// TIA Portal V17 export
// export: Created 2024-09-04T07:03:07.1988734Z, ExportSetting None, DisplayName Totally Integrated Automation Portal, DisplayVersion V17 Update 7, DisplayName TIA Portal Openness, DisplayVersion V17 Update 7, DisplayName TIA Portal Version Control Interface, DisplayVersion V17, DisplayName SINAMICS Startdrive Advanced, DisplayVersion V17 SP2, DisplayName SINAMICS Startdrive G110M, G120, G120C, G120D, G120P, G115D, DisplayVersion V17 SP2, DisplayName SINAMICS Startdrive G130, G150, S120, S150, SINAMICS MV, S210, DisplayVersion V17 SP2, DisplayName STEP 7 Professional, DisplayVersion V17 Update 7, DisplayName STEP 7 Safety, DisplayVersion V17 Update 6, DisplayName WinCC Professional, DisplayVersion V17 Update 7
FUNCTION_BLOCK "fbMain"   // FB5, LAD
{ S7_Optimized_Access := 'TRUE' }
// IO processing block reads in the thermocouple and pressure transmitter readings into the program and outputs the valve control values. 
// 
// Recipe assignment waits for input from the HMI to assign recipes to each press. 
// 
// Press control FBs manage the sequencer and valve position control.
// stored: MemoryReserve 100, SetENOAutomatically false
   VAR
      iRecipeToLoad { S7_SetPoint := 'True'} : Int;
   END_VAR
   VAR CONSTANT
      iMode_ForceOpen : Int := 2;
   END_VAR
BEGIN

REGION Network 1: FB: Input/Output Processing
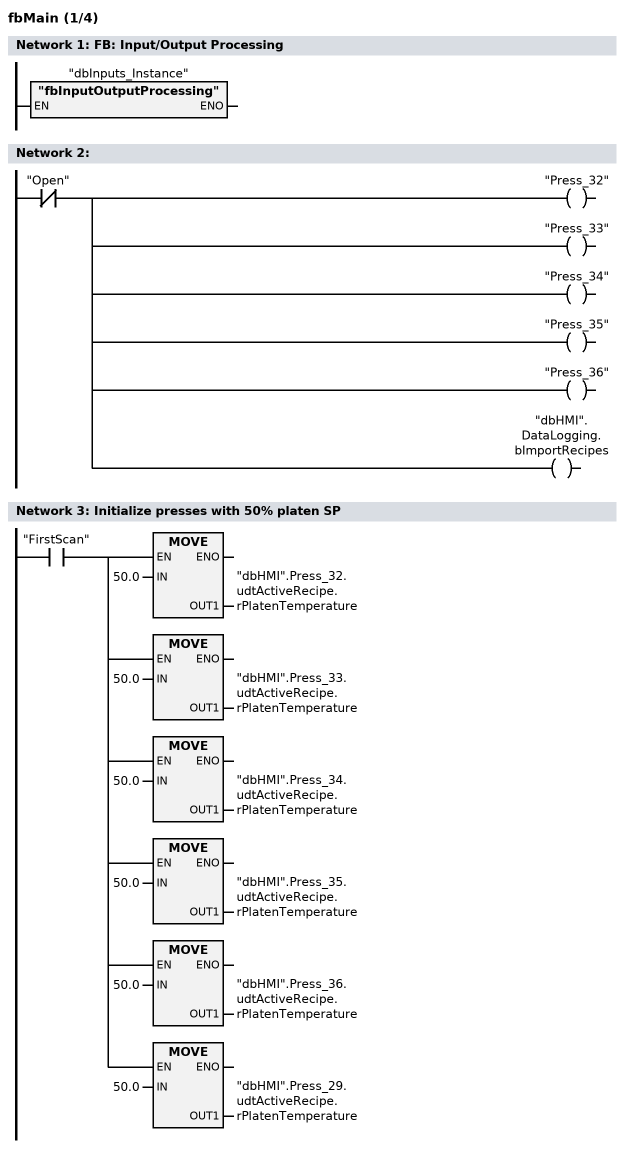
   RUNG wire#powerrail
      "dbInputs_Instance"()
   END_RUNG
   // the same network as SCL:
   "dbInputs_Instance"();   // "fbInputOutputProcessing"
END_REGION

REGION Network 2
   RUNG wire#powerrail
      I_Contact( "Open" )
      wire#w1
      Coil( "Press_32" )
   END_RUNG
   RUNG wire#w1
      Coil( "Press_33" )
   END_RUNG
   RUNG wire#w1
      Coil( "Press_34" )
   END_RUNG
   RUNG wire#w1
      Coil( "Press_35" )
   END_RUNG
   RUNG wire#w1
      Coil( "Press_36" )
   END_RUNG
   RUNG wire#w1
      Coil( "dbHMI".DataLogging.bImportRecipes )
   END_RUNG
   // the same network as SCL:
   "Press_32" := NOT "Open";
   "Press_33" := NOT "Open";
   "Press_34" := NOT "Open";
   "Press_35" := NOT "Open";
   "Press_36" := NOT "Open";
   "dbHMI".DataLogging.bImportRecipes := NOT "Open";
END_REGION

REGION Network 3: Initialize presses with 50% platen SP
   RUNG wire#powerrail
      Contact( "FirstScan" )
      wire#w1
      Move(in := 50.0, out1 => "dbHMI".Press_32.udtActiveRecipe.rPlatenTemperature)
   END_RUNG
   RUNG wire#w1
      { S7_GenerateENO := "TRUE" } Move(in := 50.0, out1 => "dbHMI".Press_33.udtActiveRecipe.rPlatenTemperature)
   END_RUNG
   RUNG wire#w1
      { S7_GenerateENO := "TRUE" } Move(in := 50.0, out1 => "dbHMI".Press_34.udtActiveRecipe.rPlatenTemperature)
   END_RUNG
   RUNG wire#w1
      { S7_GenerateENO := "TRUE" } Move(in := 50.0, out1 => "dbHMI".Press_35.udtActiveRecipe.rPlatenTemperature)
   END_RUNG
   RUNG wire#w1
      { S7_GenerateENO := "TRUE" } Move(in := 50.0, out1 => "dbHMI".Press_36.udtActiveRecipe.rPlatenTemperature)
   END_RUNG
   RUNG wire#w1
      { S7_GenerateENO := "TRUE" } Move(in := 50.0, out1 => "dbHMI".Press_29.udtActiveRecipe.rPlatenTemperature)
   END_RUNG
   // the same network as SCL:
   IF "FirstScan" THEN
       "dbHMI".Press_32.udtActiveRecipe.rPlatenTemperature := 50.0;
       "dbHMI".Press_33.udtActiveRecipe.rPlatenTemperature := 50.0;
       "dbHMI".Press_34.udtActiveRecipe.rPlatenTemperature := 50.0;
       "dbHMI".Press_35.udtActiveRecipe.rPlatenTemperature := 50.0;
       "dbHMI".Press_36.udtActiveRecipe.rPlatenTemperature := 50.0;
       "dbHMI".Press_29.udtActiveRecipe.rPlatenTemperature := 50.0;
   END_IF;
END_REGION

REGION Network 4: Initialize all presses to force open mode
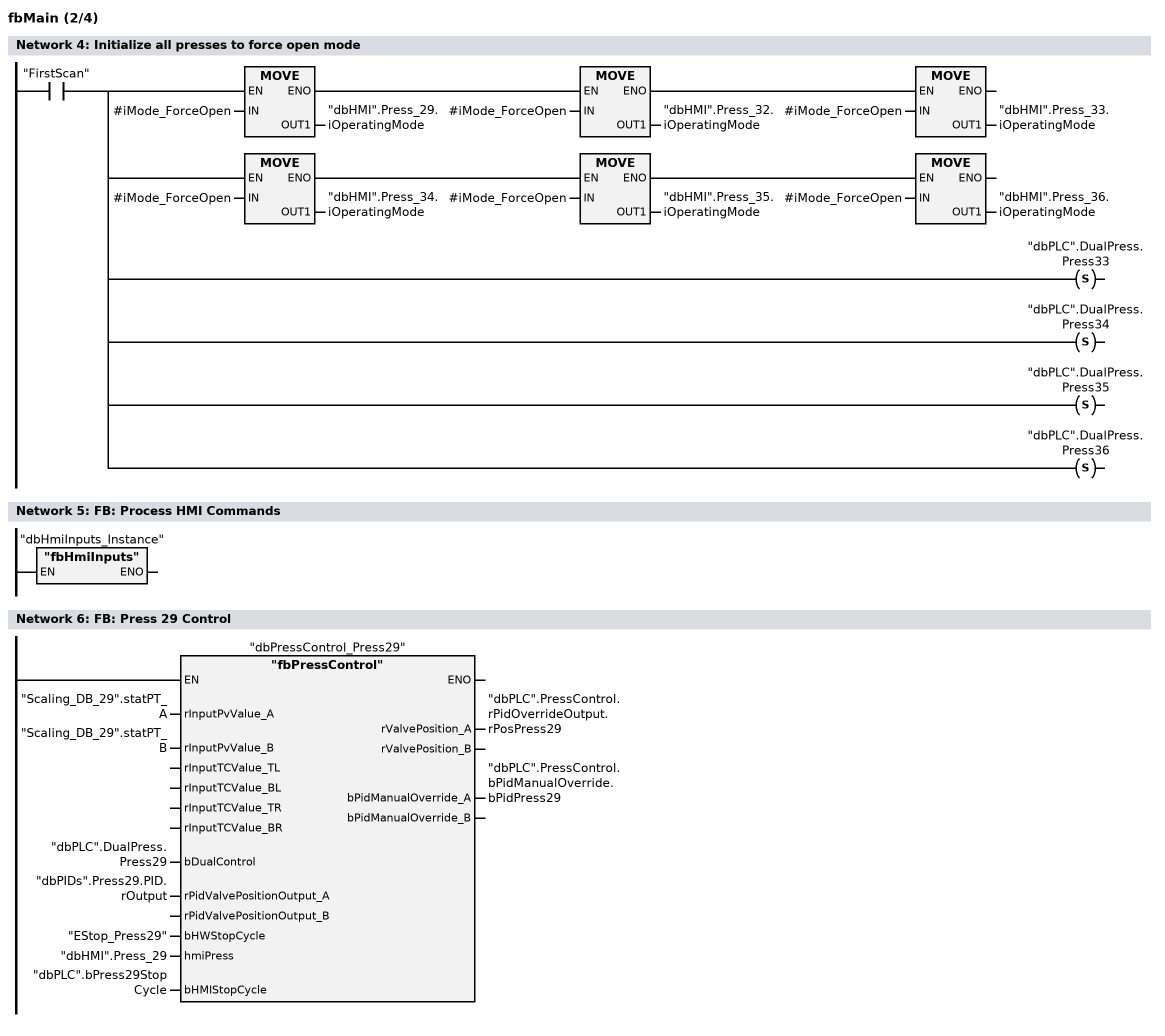
   RUNG wire#powerrail
      Contact( "FirstScan" )
      wire#w1
      { S7_GenerateENO := "TRUE" } Move(in := #iMode_ForceOpen, out1 => "dbHMI".Press_29.iOperatingMode)
      { S7_GenerateENO := "TRUE" } Move(in := #iMode_ForceOpen, out1 => "dbHMI".Press_32.iOperatingMode)
      { S7_GenerateENO := "TRUE" } Move(in := #iMode_ForceOpen, out1 => "dbHMI".Press_33.iOperatingMode)
   END_RUNG
   RUNG wire#w1
      { S7_GenerateENO := "TRUE" } Move(in := #iMode_ForceOpen, out1 => "dbHMI".Press_34.iOperatingMode)
      { S7_GenerateENO := "TRUE" } Move(in := #iMode_ForceOpen, out1 => "dbHMI".Press_35.iOperatingMode)
      { S7_GenerateENO := "TRUE" } Move(in := #iMode_ForceOpen, out1 => "dbHMI".Press_36.iOperatingMode)
   END_RUNG
   RUNG wire#w1
      S_Coil( "dbPLC".DualPress.Press33 )
   END_RUNG
   RUNG wire#w1
      S_Coil( "dbPLC".DualPress.Press34 )
   END_RUNG
   RUNG wire#w1
      S_Coil( "dbPLC".DualPress.Press35 )
   END_RUNG
   RUNG wire#w1
      S_Coil( "dbPLC".DualPress.Press36 )
   END_RUNG
   // the same network as SCL:
   // ENO of a box is taken as its EN; it also drops when the box reports an error
   IF "FirstScan" THEN
       "dbHMI".Press_29.iOperatingMode := #iMode_ForceOpen;
       "dbHMI".Press_32.iOperatingMode := #iMode_ForceOpen;
       "dbHMI".Press_33.iOperatingMode := #iMode_ForceOpen;
       "dbHMI".Press_34.iOperatingMode := #iMode_ForceOpen;
       "dbHMI".Press_35.iOperatingMode := #iMode_ForceOpen;
       "dbHMI".Press_36.iOperatingMode := #iMode_ForceOpen;
       "dbPLC".DualPress.Press33 := TRUE;
       "dbPLC".DualPress.Press34 := TRUE;
       "dbPLC".DualPress.Press35 := TRUE;
       "dbPLC".DualPress.Press36 := TRUE;
   END_IF;
END_REGION

REGION Network 5: FB: Process HMI Commands
   RUNG wire#powerrail
      "dbHmiInputs_Instance"()
   END_RUNG
   // the same network as SCL:
   "dbHmiInputs_Instance"();   // "fbHmiInputs"
END_REGION

REGION Network 6: FB: Press 29 Control
   RUNG wire#powerrail
      "dbPressControl_Press29"(rInputPvValue_A := "Scaling_DB_29".statPT_A, rInputPvValue_B := "Scaling_DB_29".statPT_B, rInputTCValue_TL :=, rInputTCValue_BL :=, rInputTCValue_TR :=, rInputTCValue_BR :=, bDualControl := "dbPLC".DualPress.Press29, rPidValvePositionOutput_A := "dbPIDs".Press29.PID.rOutput, rPidValvePositionOutput_B :=, bHWStopCycle := "EStop_Press29", hmiPress := "dbHMI".Press_29, bHMIStopCycle := "dbPLC".bPress29StopCycle, rValvePosition_A => "dbPLC".PressControl.rPidOverrideOutput.rPosPress29, rValvePosition_B =>, bPidManualOverride_A => "dbPLC".PressControl.bPidManualOverride.bPidPress29, bPidManualOverride_B =>)
   END_RUNG
   // the same network as SCL:
   "dbPressControl_Press29"(rInputPvValue_A := "Scaling_DB_29".statPT_A,   // "fbPressControl"
                           rInputPvValue_B := "Scaling_DB_29".statPT_B,
                           bDualControl := "dbPLC".DualPress.Press29,
                           rPidValvePositionOutput_A := "dbPIDs".Press29.PID.rOutput,
                           bHWStopCycle := "EStop_Press29",
                           hmiPress := "dbHMI".Press_29,
                           bHMIStopCycle := "dbPLC".bPress29StopCycle,
                           rValvePosition_A => "dbPLC".PressControl.rPidOverrideOutput.rPosPress29,
                           bPidManualOverride_A => "dbPLC".PressControl.bPidManualOverride.bPidPress29);
END_REGION

REGION Network 7: FB: Press 32 Control
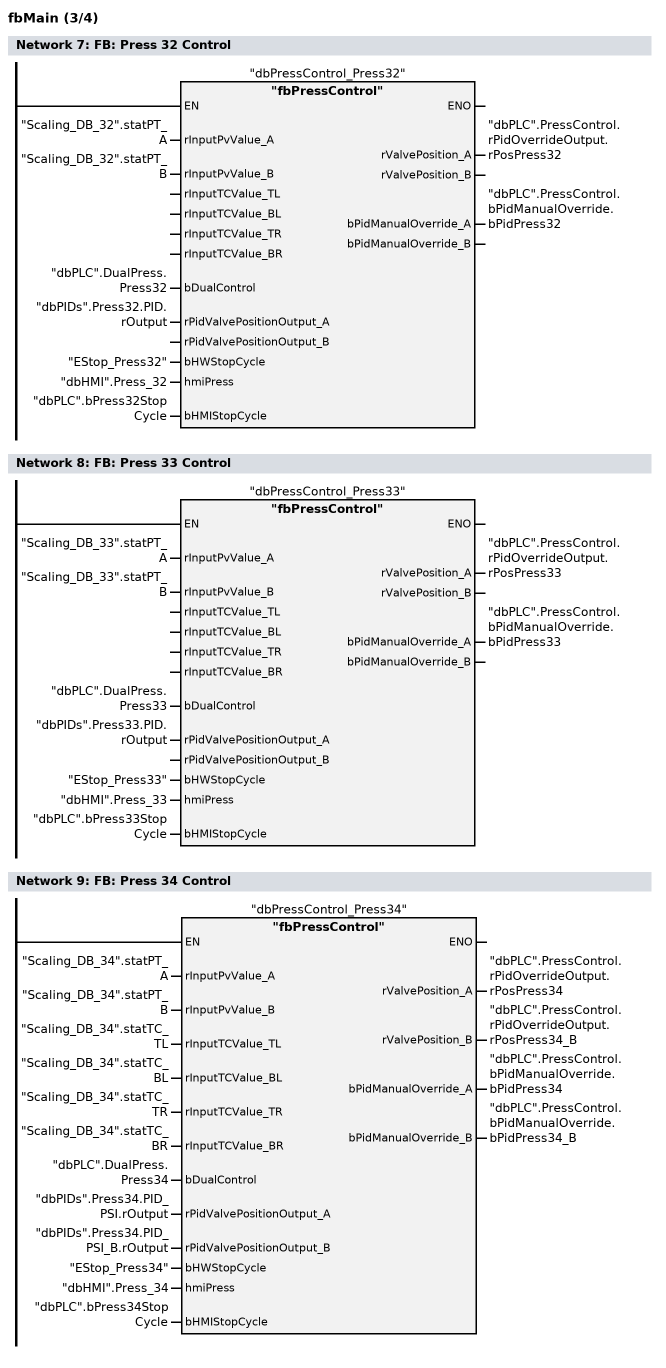
   RUNG wire#powerrail
      "dbPressControl_Press32"(rInputPvValue_A := "Scaling_DB_32".statPT_A, rInputPvValue_B := "Scaling_DB_32".statPT_B, rInputTCValue_TL :=, rInputTCValue_BL :=, rInputTCValue_TR :=, rInputTCValue_BR :=, bDualControl := "dbPLC".DualPress.Press32, rPidValvePositionOutput_A := "dbPIDs".Press32.PID.rOutput, rPidValvePositionOutput_B :=, bHWStopCycle := "EStop_Press32", hmiPress := "dbHMI".Press_32, bHMIStopCycle := "dbPLC".bPress32StopCycle, rValvePosition_A => "dbPLC".PressControl.rPidOverrideOutput.rPosPress32, rValvePosition_B =>, bPidManualOverride_A => "dbPLC".PressControl.bPidManualOverride.bPidPress32, bPidManualOverride_B =>)
   END_RUNG
   // the same network as SCL:
   "dbPressControl_Press32"(rInputPvValue_A := "Scaling_DB_32".statPT_A,   // "fbPressControl"
                           rInputPvValue_B := "Scaling_DB_32".statPT_B,
                           bDualControl := "dbPLC".DualPress.Press32,
                           rPidValvePositionOutput_A := "dbPIDs".Press32.PID.rOutput,
                           bHWStopCycle := "EStop_Press32",
                           hmiPress := "dbHMI".Press_32,
                           bHMIStopCycle := "dbPLC".bPress32StopCycle,
                           rValvePosition_A => "dbPLC".PressControl.rPidOverrideOutput.rPosPress32,
                           bPidManualOverride_A => "dbPLC".PressControl.bPidManualOverride.bPidPress32);
END_REGION

REGION Network 8: FB: Press 33 Control
   RUNG wire#powerrail
      "dbPressControl_Press33"(rInputPvValue_A := "Scaling_DB_33".statPT_A, rInputPvValue_B := "Scaling_DB_33".statPT_B, rInputTCValue_TL :=, rInputTCValue_BL :=, rInputTCValue_TR :=, rInputTCValue_BR :=, bDualControl := "dbPLC".DualPress.Press33, rPidValvePositionOutput_A := "dbPIDs".Press33.PID.rOutput, rPidValvePositionOutput_B :=, bHWStopCycle := "EStop_Press33", hmiPress := "dbHMI".Press_33, bHMIStopCycle := "dbPLC".bPress33StopCycle, rValvePosition_A => "dbPLC".PressControl.rPidOverrideOutput.rPosPress33, rValvePosition_B =>, bPidManualOverride_A => "dbPLC".PressControl.bPidManualOverride.bPidPress33, bPidManualOverride_B =>)
   END_RUNG
   // the same network as SCL:
   "dbPressControl_Press33"(rInputPvValue_A := "Scaling_DB_33".statPT_A,   // "fbPressControl"
                           rInputPvValue_B := "Scaling_DB_33".statPT_B,
                           bDualControl := "dbPLC".DualPress.Press33,
                           rPidValvePositionOutput_A := "dbPIDs".Press33.PID.rOutput,
                           bHWStopCycle := "EStop_Press33",
                           hmiPress := "dbHMI".Press_33,
                           bHMIStopCycle := "dbPLC".bPress33StopCycle,
                           rValvePosition_A => "dbPLC".PressControl.rPidOverrideOutput.rPosPress33,
                           bPidManualOverride_A => "dbPLC".PressControl.bPidManualOverride.bPidPress33);
END_REGION

REGION Network 9: FB: Press 34 Control
   RUNG wire#powerrail
      "dbPressControl_Press34"(rInputPvValue_A := "Scaling_DB_34".statPT_A, rInputPvValue_B := "Scaling_DB_34".statPT_B, rInputTCValue_TL := "Scaling_DB_34".statTC_TL, rInputTCValue_BL := "Scaling_DB_34".statTC_BL, rInputTCValue_TR := "Scaling_DB_34".statTC_TR, rInputTCValue_BR := "Scaling_DB_34".statTC_BR, bDualControl := "dbPLC".DualPress.Press34, rPidValvePositionOutput_A := "dbPIDs".Press34.PID_PSI.rOutput, rPidValvePositionOutput_B := "dbPIDs".Press34.PID_PSI_B.rOutput, bHWStopCycle := "EStop_Press34", hmiPress := "dbHMI".Press_34, bHMIStopCycle := "dbPLC".bPress34StopCycle, rValvePosition_A => "dbPLC".PressControl.rPidOverrideOutput.rPosPress34, rValvePosition_B => "dbPLC".PressControl.rPidOverrideOutput.rPosPress34_B, bPidManualOverride_A => "dbPLC".PressControl.bPidManualOverride.bPidPress34, bPidManualOverride_B => "dbPLC".PressControl.bPidManualOverride.bPidPress34_B)
   END_RUNG
   // the same network as SCL:
   "dbPressControl_Press34"(rInputPvValue_A := "Scaling_DB_34".statPT_A,   // "fbPressControl"
                           rInputPvValue_B := "Scaling_DB_34".statPT_B,
                           rInputTCValue_TL := "Scaling_DB_34".statTC_TL,
                           rInputTCValue_BL := "Scaling_DB_34".statTC_BL,
                           rInputTCValue_TR := "Scaling_DB_34".statTC_TR,
                           rInputTCValue_BR := "Scaling_DB_34".statTC_BR,
                           bDualControl := "dbPLC".DualPress.Press34,
                           rPidValvePositionOutput_A := "dbPIDs".Press34.PID_PSI.rOutput,
                           rPidValvePositionOutput_B := "dbPIDs".Press34.PID_PSI_B.rOutput,
                           bHWStopCycle := "EStop_Press34",
                           hmiPress := "dbHMI".Press_34,
                           bHMIStopCycle := "dbPLC".bPress34StopCycle,
                           rValvePosition_A => "dbPLC".PressControl.rPidOverrideOutput.rPosPress34,
                           rValvePosition_B => "dbPLC".PressControl.rPidOverrideOutput.rPosPress34_B,
                           bPidManualOverride_A => "dbPLC".PressControl.bPidManualOverride.bPidPress34,
                           bPidManualOverride_B => "dbPLC".PressControl.bPidManualOverride.bPidPress34_B);
END_REGION

REGION Network 10: FB: Press 35 Control
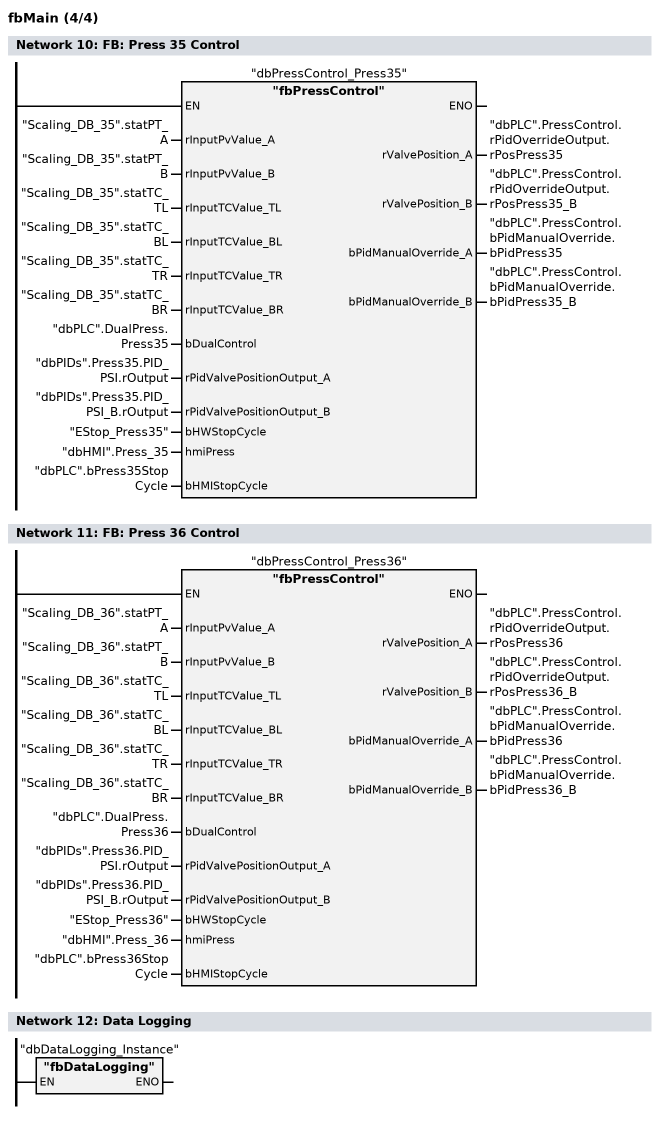
   RUNG wire#powerrail
      "dbPressControl_Press35"(rInputPvValue_A := "Scaling_DB_35".statPT_A, rInputPvValue_B := "Scaling_DB_35".statPT_B, rInputTCValue_TL := "Scaling_DB_35".statTC_TL, rInputTCValue_BL := "Scaling_DB_35".statTC_BL, rInputTCValue_TR := "Scaling_DB_35".statTC_TR, rInputTCValue_BR := "Scaling_DB_35".statTC_BR, bDualControl := "dbPLC".DualPress.Press35, rPidValvePositionOutput_A := "dbPIDs".Press35.PID_PSI.rOutput, rPidValvePositionOutput_B := "dbPIDs".Press35.PID_PSI_B.rOutput, bHWStopCycle := "EStop_Press35", hmiPress := "dbHMI".Press_35, bHMIStopCycle := "dbPLC".bPress35StopCycle, rValvePosition_A => "dbPLC".PressControl.rPidOverrideOutput.rPosPress35, rValvePosition_B => "dbPLC".PressControl.rPidOverrideOutput.rPosPress35_B, bPidManualOverride_A => "dbPLC".PressControl.bPidManualOverride.bPidPress35, bPidManualOverride_B => "dbPLC".PressControl.bPidManualOverride.bPidPress35_B)
   END_RUNG
   // the same network as SCL:
   "dbPressControl_Press35"(rInputPvValue_A := "Scaling_DB_35".statPT_A,   // "fbPressControl"
                           rInputPvValue_B := "Scaling_DB_35".statPT_B,
                           rInputTCValue_TL := "Scaling_DB_35".statTC_TL,
                           rInputTCValue_BL := "Scaling_DB_35".statTC_BL,
                           rInputTCValue_TR := "Scaling_DB_35".statTC_TR,
                           rInputTCValue_BR := "Scaling_DB_35".statTC_BR,
                           bDualControl := "dbPLC".DualPress.Press35,
                           rPidValvePositionOutput_A := "dbPIDs".Press35.PID_PSI.rOutput,
                           rPidValvePositionOutput_B := "dbPIDs".Press35.PID_PSI_B.rOutput,
                           bHWStopCycle := "EStop_Press35",
                           hmiPress := "dbHMI".Press_35,
                           bHMIStopCycle := "dbPLC".bPress35StopCycle,
                           rValvePosition_A => "dbPLC".PressControl.rPidOverrideOutput.rPosPress35,
                           rValvePosition_B => "dbPLC".PressControl.rPidOverrideOutput.rPosPress35_B,
                           bPidManualOverride_A => "dbPLC".PressControl.bPidManualOverride.bPidPress35,
                           bPidManualOverride_B => "dbPLC".PressControl.bPidManualOverride.bPidPress35_B);
END_REGION

REGION Network 11: FB: Press 36 Control
   RUNG wire#powerrail
      "dbPressControl_Press36"(rInputPvValue_A := "Scaling_DB_36".statPT_A, rInputPvValue_B := "Scaling_DB_36".statPT_B, rInputTCValue_TL := "Scaling_DB_36".statTC_TL, rInputTCValue_BL := "Scaling_DB_36".statTC_BL, rInputTCValue_TR := "Scaling_DB_36".statTC_TR, rInputTCValue_BR := "Scaling_DB_36".statTC_BR, bDualControl := "dbPLC".DualPress.Press36, rPidValvePositionOutput_A := "dbPIDs".Press36.PID_PSI.rOutput, rPidValvePositionOutput_B := "dbPIDs".Press36.PID_PSI_B.rOutput, bHWStopCycle := "EStop_Press36", hmiPress := "dbHMI".Press_36, bHMIStopCycle := "dbPLC".bPress36StopCycle, rValvePosition_A => "dbPLC".PressControl.rPidOverrideOutput.rPosPress36, rValvePosition_B => "dbPLC".PressControl.rPidOverrideOutput.rPosPress36_B, bPidManualOverride_A => "dbPLC".PressControl.bPidManualOverride.bPidPress36, bPidManualOverride_B => "dbPLC".PressControl.bPidManualOverride.bPidPress36_B)
   END_RUNG
   // the same network as SCL:
   "dbPressControl_Press36"(rInputPvValue_A := "Scaling_DB_36".statPT_A,   // "fbPressControl"
                           rInputPvValue_B := "Scaling_DB_36".statPT_B,
                           rInputTCValue_TL := "Scaling_DB_36".statTC_TL,
                           rInputTCValue_BL := "Scaling_DB_36".statTC_BL,
                           rInputTCValue_TR := "Scaling_DB_36".statTC_TR,
                           rInputTCValue_BR := "Scaling_DB_36".statTC_BR,
                           bDualControl := "dbPLC".DualPress.Press36,
                           rPidValvePositionOutput_A := "dbPIDs".Press36.PID_PSI.rOutput,
                           rPidValvePositionOutput_B := "dbPIDs".Press36.PID_PSI_B.rOutput,
                           bHWStopCycle := "EStop_Press36",
                           hmiPress := "dbHMI".Press_36,
                           bHMIStopCycle := "dbPLC".bPress36StopCycle,
                           rValvePosition_A => "dbPLC".PressControl.rPidOverrideOutput.rPosPress36,
                           rValvePosition_B => "dbPLC".PressControl.rPidOverrideOutput.rPosPress36_B,
                           bPidManualOverride_A => "dbPLC".PressControl.bPidManualOverride.bPidPress36,
                           bPidManualOverride_B => "dbPLC".PressControl.bPidManualOverride.bPidPress36_B);
END_REGION

REGION Network 12: Data Logging
   RUNG wire#powerrail
      "dbDataLogging_Instance"()
   END_RUNG
   // the same network as SCL:
   "dbDataLogging_Instance"();   // "fbDataLogging"
END_REGION
END_FUNCTION_BLOCK
